{attribute addProperty BoxType "ELX4181-0000-0016"}
{attribute addProperty Id "Ch_1Ch_1_10CBEF651620WcStateAT %I*WcState_64F6A8C6810InfoDataAT %I*InfoData_275E3363128160"}
{attribute addProperty CRC "152658471"}
{attribute addProperty SizeInBites "152"}
{attribute addProperty SizeInBytes "19"}
TYPE ELX4181_E6374D8B :
STRUCT
	{attribute addProperty Name "Ch_1"}
	Ch_1 : Ch_1_10CBEF65;
	{attribute addProperty Name "WcState"}
	WcState : WcState_64F6A8C6;
	{attribute addProperty Name "InfoData"}
	InfoData : InfoData_275E3363;
END_STRUCT
END_TYPE

(* stored: Version 1.2.0.0, ProductVersion 3.1.4024.9
   DUT ELX4181_E6374D8B: Id {9ee56157-2f81-4abb-b9ea-b37bdfdf29b7} *)
